(* CoDeSys 2.3 export: TCWIESENRAIN23.EXP *)
(* Libraries: STANDARD.LIB 5.6.98 12:03:02, TcBase.lib 14.5.09 12:14:08, TcEtherCAT.lib 8.3.12 17:06:42, TcSUPS.lib 22.3.10 13:59:22, TcSystem.lib 27.2.12 15:08:36, TcUtilities.lib 10.1.13 20:12:12 *)

(* Task configuration *)
TASK Standard (PRIORITY := 1, INTERVAL := T#10ms);
MAIN
END_TASK
TASK Fast (PRIORITY := 0, INTERVAL := T#1ms);
IO_FAST
END_TASK

(* Global variable list: TwinCAT_Configuration *)
(* Generated automatically by TwinCAT - (read only) *)
VAR_CONFIG
	IO_FAST.uiStateCX5000 AT %IB0 : UINT;
	IO_FAST.uiControlCX5000 AT %QB0 : UINT;
	IO_FAST.iVoltagePhase1 AT %IB2 : ARRAY [0..9] OF INT;	(*  ~ {LinkedWith:TIID^KG-HV A1 X001 (EtherCAT)^KG-HV A35^KG-HV A18^L1 Voltage Samples^U1 SAMPLES} *)
	IO_FAST.iVoltagePhase2 AT %IB22 : ARRAY [0..9] OF INT;	(*  ~ {LinkedWith:TIID^KG-HV A1 X001 (EtherCAT)^KG-HV A35^KG-HV A18^L2 Voltage Samples^U2 SAMPLES} *)
	IO_FAST.iVoltagePhase3 AT %IB42 : ARRAY [0..9] OF INT;	(*  ~ {LinkedWith:TIID^KG-HV A1 X001 (EtherCAT)^KG-HV A35^KG-HV A18^L3 Voltage Samples^U3 SAMPLES} *)
	IO_FAST.uliStartTimeNextLatch AT %IB62 : ARRAY [0..1] OF UDINT;	(*  ~ {LinkedWith:TIID^KG-HV A1 X001 (EtherCAT)^KG-HV A35^KG-HV A18^AI Timestamp NextSync1Time^StartTimeNextLatch} *)
	IO_FAST.bWcState AT %IX72.0 : BOOL;	(*  ~ {LinkedWith:TIID^KG-HV A1 X001 (EtherCAT)^KG-HV A35^KG-HV A18^WcState^WcState} *)
	IO_FAST.fbA28CH1.bRelay AT %QX2.0 : BOOL;	(*  ~ {LinkedWith:TIID^KG-HV A1 K-Bus^KG-HV A1^KG-HV A28^Kanal 1^Ausgang} *)
	IO_FAST.fbA28CH2.bRelay AT %QX2.1 : BOOL;	(*  ~ {LinkedWith:TIID^KG-HV A1 K-Bus^KG-HV A1^KG-HV A28^Kanal 2^Ausgang} *)
	IO_FAST.fbA29CH1.bRelay AT %QX2.2 : BOOL;	(*  ~ {LinkedWith:TIID^KG-HV A1 K-Bus^KG-HV A1^KG-HV A29^Kanal 1^Ausgang} *)
	IO_FAST.fbA29CH2.bRelay AT %QX2.3 : BOOL;	(*  ~ {LinkedWith:TIID^KG-HV A1 K-Bus^KG-HV A1^KG-HV A29^Kanal 2^Ausgang} *)
	IO_FAST.fbA30CH1.bRelay AT %QX2.4 : BOOL;	(*  ~ {LinkedWith:TIID^KG-HV A1 K-Bus^KG-HV A1^KG-HV A30^Kanal 1^Ausgang} *)
	IO_FAST.fbA30CH2.bRelay AT %QX2.5 : BOOL;	(*  ~ {LinkedWith:TIID^KG-HV A1 K-Bus^KG-HV A1^KG-HV A30^Kanal 2^Ausgang} *)
	IO_FAST.fbA31CH1.bRelay AT %QX2.6 : BOOL;	(*  ~ {LinkedWith:TIID^KG-HV A1 K-Bus^KG-HV A1^KG-HV A31^Kanal 1^Ausgang} *)
	IO_FAST.fbA31CH2.bRelay AT %QX2.7 : BOOL;	(*  ~ {LinkedWith:TIID^KG-HV A1 K-Bus^KG-HV A1^KG-HV A31^Kanal 2^Ausgang} *)
	IO_FAST.fbA32CH1.bRelay AT %QX3.0 : BOOL;	(*  ~ {LinkedWith:TIID^KG-HV A1 K-Bus^KG-HV A1^KG-HV A32^Kanal 1^Ausgang} *)
	IO_FAST.fbA32CH2.bRelay AT %QX3.1 : BOOL;	(*  ~ {LinkedWith:TIID^KG-HV A1 K-Bus^KG-HV A1^KG-HV A32^Kanal 2^Ausgang} *)
	IO_FAST.fbA20CH1.bRelay AT %QX3.2 : BOOL;	(*  ~ {LinkedWith:TIID^KG-HV A1 K-Bus^KG-HV A1^KG-HV A20^Kanal 1^KG-Gang Lampe} *)
	IO_FAST.fbA20CH2.bRelay AT %QX3.3 : BOOL;	(*  ~ {LinkedWith:TIID^KG-HV A1 K-Bus^KG-HV A1^KG-HV A20^Kanal 2^KG-EG-Stiege Lampe} *)
	IO_FAST.fbA21CH1.bRelay AT %QX3.4 : BOOL;	(*  ~ {LinkedWith:TIID^KG-HV A1 K-Bus^KG-HV A1^KG-HV A21^Kanal 1^Lager Lampe} *)
	IO_FAST.fbA21CH2.bRelay AT %QX3.5 : BOOL;	(*  ~ {LinkedWith:TIID^KG-HV A1 K-Bus^KG-HV A1^KG-HV A21^Kanal 2^Ausgang} *)
	IO_FAST.fbA23CH1.bRelay AT %QX3.6 : BOOL;	(*  ~ {LinkedWith:TIID^KG-HV A1 K-Bus^KG-HV A1^KG-HV A23^Kanal 1^Heizen Lampe} *)
	IO_FAST.fbA23CH2.bRelay AT %QX3.7 : BOOL;	(*  ~ {LinkedWith:TIID^KG-HV A1 K-Bus^KG-HV A1^KG-HV A23^Kanal 2^WaschenS Lampe} *)
	IO_FAST.fbA24CH1.bRelay AT %QX4.0 : BOOL;	(*  ~ {LinkedWith:TIID^KG-HV A1 K-Bus^KG-HV A1^KG-HV A24^Kanal 1^WaschenN Lampe} *)
	IO_FAST.fbA24CH2.bRelay AT %QX4.1 : BOOL;	(*  ~ {LinkedWith:TIID^KG-HV A1 K-Bus^KG-HV A1^KG-HV A24^Kanal 2^HobbyN Lampe} *)
	IO_FAST.fbA25CH1.bRelay AT %QX4.2 : BOOL;	(*  ~ {LinkedWith:TIID^KG-HV A1 K-Bus^KG-HV A1^KG-HV A25^Kanal 1^Vorrat Lampe} *)
	IO_FAST.fbA25CH2.bRelay AT %QX4.3 : BOOL;	(*  ~ {LinkedWith:TIID^KG-HV A1 K-Bus^KG-HV A1^KG-HV A25^Kanal 2^HobbyS Lampe} *)
	IO_FAST.fbA26CH1.bRelay AT %QX4.4 : BOOL;	(*  ~ {LinkedWith:TIID^KG-HV A1 K-Bus^KG-HV A1^KG-HV A26^Kanal 1^Ausgang} *)
	IO_FAST.fbA26CH2.bRelay AT %QX4.5 : BOOL;	(*  ~ {LinkedWith:TIID^KG-HV A1 K-Bus^KG-HV A1^KG-HV A26^Kanal 2^Ausgang} *)
	IO_FAST.fbA38OGCH1.bRelay AT %QX4.6 : BOOL;
	IO_FAST.fbA38OGCH2.bRelay AT %QX4.7 : BOOL;
	IO_FAST.fbA41OGCH1.bRelay AT %QX5.0 : BOOL;
	IO_FAST.fbA41OGCH2.bRelay AT %QX5.1 : BOOL;
	IO_FAST.fbA43OGCH1.bRelay AT %QX5.2 : BOOL;
	IO_FAST.fbA43OGCH2.bRelay AT %QX5.3 : BOOL;
	IO_FAST.fbA44OGCH1.bRelay AT %QX5.4 : BOOL;
	IO_FAST.fbA44OGCH2.bRelay AT %QX5.5 : BOOL;
	IO_FAST.fbA45OGCH1.bRelay AT %QX5.6 : BOOL;
	IO_FAST.fbA45OGCH2.bRelay AT %QX5.7 : BOOL;
	IO_FAST.fbA48OGCH1.bRelay AT %QX6.0 : BOOL;
	IO_FAST.fbA48OGCH2.bRelay AT %QX6.1 : BOOL;
	IO_FAST.fbA49OGCH1.bRelay AT %QX6.2 : BOOL;
	IO_FAST.fbA49OGCH2.bRelay AT %QX6.3 : BOOL;
	IO_FAST.fbA50OGCH1.bRelay AT %QX6.4 : BOOL;
	IO_FAST.fbA50OGCH2.bRelay AT %QX6.5 : BOOL;
	IO_FAST.fbA52OGCH1.bRelay AT %QX6.6 : BOOL;
	IO_FAST.fbA52OGCH2.bRelay AT %QX6.7 : BOOL;
	IO_FAST.fbA53OGCH1.bRelay AT %QX7.0 : BOOL;
	IO_FAST.fbA53OGCH2.bRelay AT %QX7.1 : BOOL;
	IO_FAST.fbA55OGCH1.bRelay AT %QX7.2 : BOOL;
	IO_FAST.fbA55OGCH2.bRelay AT %QX7.3 : BOOL;
	IO_FAST.fbA56OGCH1.bRelay AT %QX7.4 : BOOL;
	IO_FAST.fbA56OGCH2.bRelay AT %QX7.5 : BOOL;
	IO_FAST.fbA57OGCH1.bRelay AT %QX7.6 : BOOL;
	IO_FAST.fbA57OGCH2.bRelay AT %QX7.7 : BOOL;
	IO_FAST.fbA15OGCH1.bRelay AT %QX8.0 : BOOL;
	IO_FAST.fbA15OGCH2.bRelay AT %QX8.1 : BOOL;
	IO_FAST.fbA17OGCH1.bRelay AT %QX8.2 : BOOL;
	IO_FAST.fbA17OGCH2.bRelay AT %QX8.3 : BOOL;
	IO_FAST.fbA18OGCH1.bRelay AT %QX8.4 : BOOL;
	IO_FAST.fbA18OGCH2.bRelay AT %QX8.5 : BOOL;
	IO_FAST.fbA19OGCH1.bRelay AT %QX8.6 : BOOL;
	IO_FAST.fbA19OGCH2.bRelay AT %QX8.7 : BOOL;
	IO_FAST.fbA21OGCH1.bRelay AT %QX9.0 : BOOL;
	IO_FAST.fbA21OGCH2.bRelay AT %QX9.1 : BOOL;
	IO_FAST.fbA23OGCH1.bRelay AT %QX9.2 : BOOL;
	IO_FAST.fbA23OGCH2.bRelay AT %QX9.3 : BOOL;
	IO_FAST.fbA25OGCH1.bRelay AT %QX9.4 : BOOL;
	IO_FAST.fbA25OGCH2.bRelay AT %QX9.5 : BOOL;
	IO_FAST.fbA26OGCH1.bRelay AT %QX9.6 : BOOL;
	IO_FAST.fbA26OGCH2.bRelay AT %QX9.7 : BOOL;
	IO_FAST.fbA33OGCH1.bRelay AT %QX10.0 : BOOL;
	IO_FAST.fbA33OGCH2.bRelay AT %QX10.1 : BOOL;
	IO_FAST.fbA35OGCH1.bRelay AT %QX10.2 : BOOL;
	IO_FAST.fbA35OGCH2.bRelay AT %QX10.3 : BOOL;
	IO_FAST.fbA36OGCH1.bRelay AT %QX10.4 : BOOL;
	IO_FAST.fbA36OGCH2.bRelay AT %QX10.5 : BOOL;
	IO_FAST.fbA78OGCH1.bRelay AT %QX10.6 : BOOL;
	IO_FAST.fbA78OGCH2.bRelay AT %QX10.7 : BOOL;
	IO_FAST.fbA80OGCH1.bRelay AT %QX11.0 : BOOL;
	IO_FAST.fbA80OGCH2.bRelay AT %QX11.1 : BOOL;
	MAIN._bwmKgGang AT %IX76.0 : BOOL;
	MAIN._tasterHeizen AT %IX76.1 : BOOL;
	MAIN._tasterHobbyL AT %IX76.2 : BOOL;
	MAIN._tasterHobbyR AT %IX76.3 : BOOL;
	MAIN._tasterWaschenL AT %IX76.4 : BOOL;
	MAIN._tasterWaschenR AT %IX76.5 : BOOL;
	MAIN._tasterLagerNO AT %IX76.6 : BOOL;
	MAIN._tasterLagerS AT %IX76.7 : BOOL;
	MAIN._tasterEgGangStiege AT %IX77.0 : BOOL;
	MAIN.heizenHK1.mischer AT %QB12 : INT;
	MAIN.heizenHK1.pumpe AT %QB14 : INT;
	MAIN.heizenHK2.mischer AT %QB16 : INT;
	MAIN.heizenHK2.pumpe AT %QB18 : INT;
END_VAR

(* POU MAIN, ST *)
PROGRAM MAIN
VAR
	ups: FB_S_UPS;
	toggle: FB_Toggle;

	_bwmKgGang AT %I*: BOOL; (* Ost *)
	_tasterHeizen AT %I*: BOOL; (* Sued-West *)
	_tasterHobbyL AT %I*: BOOL; (* Ost *)
	_tasterHobbyR AT %I*: BOOL; (* Ost *)
	_tasterWaschenL AT %I*: BOOL; (* West-Sued *)
	_tasterWaschenR AT %I*: BOOL; (* West-Sued *)
	_tasterLagerNO AT %I*: BOOL;
	_tasterLagerS AT %I*: BOOL;
	_tasterEgGangStiege AT %I*: BOOL; (* Nord *)

	kgGangBwm: FB_Bwm;
	kgGangLicht: FB_Light;

	heizenTaster: FB_Button;
	heizenLicht: FB_Light;
	heizenHK1: FB_Heizkreis;
	heizenHK2: FB_Heizkreis;

	hobbyLichtN: FB_Light;
	hobbyLichtS: FB_Light;

	waschenLichtN: FB_Light;
	waschenLichtS: FB_Light;

	lagerTasterNO: FB_Button;
	lagerTasterS: FB_Button;
	lagerLicht: FB_Light;

	vorratLicht: FB_Light;

	kgEgStiegeLicht: FB_Light;

END_VAR
ups();

(* input processing *)
kgGangBwm(IN := _bwmKgGang, ROOM := 'KG-Gang', LOCATION := 'Ost');
heizenTaster(IN := _tasterHeizen, ROOM := 'Heizen', LOCATION := 'Nord-West');
lagerTasterNO(IN := _tasterLagerNO, ROOM := 'Lager', LOCATION := 'Nord-Ost');
lagerTasterS(IN := _tasterLagerS, ROOM := 'Lager', LOCATION := 'Sued');

(* control *)
toggle(onTime := t#1s, offTime := t#2s);

(* output processing *)
kgGangLicht(IN := kgGangBwm.Q, PT := t#2m);
heizenLicht(IN := heizenTaster.pulseOnClick OR heizentaster.pulseOnLongpress,
	PT := t#15m,
	ROOM := 'Heizen', LOCATION := 'West|Ost');
hobbyLichtS(IN := _tasterHobbyR, PT := t#10m);
waschenLichtN(IN := _tasterWaschenR , PT := t#15m);
waschenLichtS(IN := _tasterWaschenL , PT := t#15m);
lagerLicht(IN := lagerTasterNO.pulseOnClick, FORCE := vorratLicht.Q, FORCE_ON := vorratLicht.Q, PT := t#3m);
vorratLicht(IN := lagerTasterS.pulseOnClick , PT := t#2m);
kgEgStiegeLicht(IN := _tasterEgGangStiege, PT := t#1m);

heizenHk1(soll := 24.0, vorlauf :=, ruecklauf :=);
heizenHk2(soll := 24.0, vorlauf :=, ruecklauf :=);
END_PROGRAM

(* POU FBs/FB_Toggle, ST *)
FUNCTION_BLOCK FB_Toggle
VAR_INPUT
	onTime: TIME :=  t#0.5s;
	offTime: TIME := t#1s;
END_VAR
VAR_OUTPUT
	Q: BOOL;
END_VAR
VAR
	t1: TON;
	t2: TOF;
END_VAR
t1(IN := NOT t2.Q, pt := offTime);
t2(IN := t1.Q, pt := onTime);
Q := t2.Q;
END_FUNCTION_BLOCK

(* POU FBs/FB_Bwm, ST *)
FUNCTION_BLOCK FB_Bwm
VAR_INPUT
	IN: BOOL;
	ROOM: STRING;
	LOCATION: STRING;
END_VAR
VAR_OUTPUT
	Q: BOOL;
END_VAR
Q := IN;
END_FUNCTION_BLOCK

(* POU FBs/FB_Light, ST *)
FUNCTION_BLOCK FB_Light
VAR_INPUT
	IN: BOOL;   (* on/off pulse *)
	PT: TIME;   (* auto-off aka on-time *)
	REACTION: TIME := t#1s;   (* TODO: do not change state right after statechange*)
	FORCE: BOOL;   (* if true, force output on/off, depending on FORCE_ON *)
	FORCE_ON: BOOL;   (* if false and FORCE, then force off *)
	ROOM: STRING;
	LOCATION: STRING;
END_VAR
VAR_OUTPUT RETAIN PERSISTENT
	usageTime: TIME := t#0ms;
	usageDays: UINT := 0;
	usageCounterSwitchOn: UDINT := 0;
END_VAR
VAR_OUTPUT
	Q: BOOL;
END_VAR
VAR
	viText: STRING;
	t: TOF;
	startOpTrigger: R_TRIG;
	stopOpTrigger: F_TRIG;
	opTimetracker: TIME;
	now: TIME;
END_VAR
VAR CONSTANT
	MAX_TIME: TIME := T#71582m47s295ms;
END_VAR
viText := CONCAT(ROOM, '$N');
viText := CONCAT(viText, LOCATION);

IF FORCE THEN
	IF FORCE_ON THEN
		Q := TRUE;
	ELSE
		Q := FALSE;
	END_IF
ELSE (* NOT FORCE *)
	IF IN AND t.Q THEN   (* light on and a signal *)
		(* turn off *)
		t(IN := FALSE, PT := t#0s);
	ELSIF IN AND NOT t.Q THEN   (* light off and a signal *)
		(* turn on *);
		t(IN := IN, PT := PT);
	ELSE (* timer *)
		t(IN := IN, PT := PT);
	END_IF
	Q := t.Q;
END_IF

(* record the operation time *)
startOpTrigger(CLK := Q);
stopOpTrigger(CLK := Q);
IF Q THEN
	now := TIME();
END_IF
IF startOpTrigger.Q THEN
	usageCounterSwitchOn := usageCounterSwitchOn + 1;
	opTimetracker := now;
END_IF
IF Q AND (now < opTimetracker) THEN   (* overflow *)
	usageTime := usageTime + (MAX_TIME - opTimetracker);
	opTimetracker := t#0ms;
END_IF
IF stopOpTrigger.Q THEN
	usageTime := usageTime + (now - opTimetracker);
END_IF
IF Q AND ((now - opTimetracker) > t#1s) THEN
	usageTime := usageTime + (now - opTimetracker);
	opTimetracker := now;
END_IF
IF (Q OR stopOpTrigger.Q) AND (usageTime > t#1d) THEN
	usageDays := usageDays + 1;
	usageTime := usageTime - t#1d;
END_IF
END_FUNCTION_BLOCK

(* POU FBs/FB_Button, ST *)
FUNCTION_BLOCK FB_Button
VAR_INPUT
	ROOM: STRING;
	LOCATION: STRING;
	IN: BOOL;
	LONGPRESS: TIME := t#250ms; (*read by the visualisation*)
END_VAR
VAR_OUTPUT RETAIN PERSISTENT
	isPressed: BOOL := FALSE;
	isLongpressed: BOOL := FALSE;
	isClicked: BOOL := FALSE;
	toggleOnPress: BOOL;
	toggleOnRelease: BOOL;
	toggleOnLongpress: BOOL;
	toggleOnClick: BOOL;
	usageCounterPress: UDINT; (*overall number of press events*)
	usageCounterRelease: UDINT; (*overall number of release events*)
	usageCounterLongpress: UDINT; (*overall number longpress events*)
	usageCounterClick: UDINT; (*overall number of click events*)
END_VAR
VAR_OUTPUT
	isReleased: BOOL; (*NOT isPressed*)
	pulseOnPress: BOOL;
	pulseOnRelease: BOOL;
	pulseOnLongpress: BOOL;
	pulseOnClick: BOOL;
END_VAR
VAR
	viIN: BOOL; (*written by the visualisation*)
	viText: STRING; (*read by the visualisation*)
	pTrig: R_TRIG;
	rTrig: F_TRIG;
	longpressTimer: TON;
	lTrig: R_TRIG;
	cTrig: R_TRIG;
	t1: TOF;
	t2: TOF;
	myIN: BOOL;
END_VAR
(* support VIsualisations *)
viText := CONCAT(ROOM, ' ');
viText := CONCAT(viText, LOCATION);
myIN := IN XOR viIN;

pTrig(CLK := myIN);
rTrig(CLK := myIN);
pulseOnPress := pTrig.Q;
pulseOnRelease := rTrig.Q;

longpressTimer(IN := myIN, PT := LONGPRESS);
lTrig(CLK := longpressTimer.Q);
pulseOnLongpress := ltrig.Q;
IF pulseOnLongpress AND NOT pulseOnRelease THEN
	isLongpressed := TRUE;
	usageCounterLongpress := usageCounterLongpress + 1;
	toggleOnLongpress := fToggle(toggleOnLongpress);
ELSIF pulseOnLongpress THEN
	pulseOnLongpress := FALSE;
END_IF

IF pulseOnPress THEN
	isPressed := TRUE;
	isClicked := FALSE;
	isLongpressed := FALSE;
	usageCounterPress := usageCounterPress + 1;
	toggleOnPress := fToggle(toggleOnPress);
ELSIF pulseOnRelease THEN
	isPressed := FALSE;
	IF isLongpressed THEN
		isLongpressed := FALSE;
	ELSE
		isClicked := TRUE;
		usageCounterClick := usageCounterClick + 1;
		toggleOnClick := fToggle(toggleOnClick);
	END_IF
	usageCounterRelease := usageCounterRelease + 1;
	toggleOnRelease := fToggle(toggleOnRelease);
END_IF
isReleased := NOT isPressed;

cTrig(CLK := isClicked);
pulseOnClick := cTrig.Q;
END_FUNCTION_BLOCK

(* POU Fs/fToggle, ST *)
FUNCTION fToggle : BOOL
VAR_INPUT
	IN: BOOL;
END_VAR
IF IN THEN
	fToggle := FALSE;
ELSE
	fToggle := TRUE;
END_IF
END_FUNCTION

(* POU FBs/FB_Heizkreis, ST *)
FUNCTION_BLOCK FB_Heizkreis
VAR_INPUT
	soll:REAL;
	vorlauf: REAL;
	ruecklauf: REAL;
END_VAR
VAR_OUTPUT
	mischer AT %Q*: INT;   (* 0x7FFF = 100% = 10V; 0x0000 = 0% = 0V*)
	pumpe AT %Q*: INT;   (* 0x7FFF = 100% = 10V; 0x0000 = 0% = 0V*)
END_VAR
VAR
END_VAR
mischer := 6000;
pumpe := 0;
END_FUNCTION_BLOCK

(* POU IO_FAST, ST *)
PROGRAM IO_FAST
VAR
	uiStateCX5000 AT %I*: UINT;
	uiControlCX5000 AT %Q* : UINT;
	iVoltagePhase1 AT %I* : ARRAY [0..9] OF INT;
	iVoltagePhase2 AT %I* : ARRAY [0..9] OF INT;
	iVoltagePhase3 AT %I* : ARRAY [0..9] OF INT;
	uliStartTimeNextLatch AT %I* : ARRAY [0..1] OF UDINT;
	bWcState AT %I* : BOOL;

	fbAnalyseVoltagePhase1 : FB_ANALYSE_VOLTAGE;
	fbAnalyseVoltagePhase2 : FB_ANALYSE_VOLTAGE;
	fbAnalyseVoltagePhase3 : FB_ANALYSE_VOLTAGE;
	fbA28CH1: FB_SYNC_RELAIS;
	fbA28CH2: FB_SYNC_RELAIS;
	fbA29CH1: FB_SYNC_RELAIS;
	fbA29CH2: FB_SYNC_RELAIS;
	fbA30CH1: FB_SYNC_RELAIS;
	fbA30CH2: FB_SYNC_RELAIS;
	fbA31CH1: FB_SYNC_RELAIS;
	fbA31CH2: FB_SYNC_RELAIS;
	fbA32CH1: FB_SYNC_RELAIS;
	fbA32CH2: FB_SYNC_RELAIS;
	fbA20CH1: FB_SYNC_RELAIS;
	fbA20CH2: FB_SYNC_RELAIS;
	fbA21CH1: FB_SYNC_RELAIS;
	fbA21CH2: FB_SYNC_RELAIS;
	fbA23CH1: FB_SYNC_RELAIS;
	fbA23CH2: FB_SYNC_RELAIS;
	fbA24CH1: FB_SYNC_RELAIS;
	fbA24CH2: FB_SYNC_RELAIS;
	fbA25CH1: FB_SYNC_RELAIS;
	fbA25CH2: FB_SYNC_RELAIS;
	fbA26CH1: FB_SYNC_RELAIS;
	fbA26CH2: FB_SYNC_RELAIS;
	fbA38OGCH1: FB_SYNC_RELAIS;
	fbA38OGCH2: FB_SYNC_RELAIS;
	fbA41OGCH1: FB_SYNC_RELAIS;
	fbA41OGCH2: FB_SYNC_RELAIS;
	fbA43OGCH1: FB_SYNC_RELAIS;
	fbA43OGCH2: FB_SYNC_RELAIS;
	fbA44OGCH1: FB_SYNC_RELAIS;
	fbA44OGCH2: FB_SYNC_RELAIS;
	fbA45OGCH1: FB_SYNC_RELAIS;
	fbA45OGCH2: FB_SYNC_RELAIS;
	fbA48OGCH1: FB_SYNC_RELAIS;
	fbA48OGCH2: FB_SYNC_RELAIS;
	fbA49OGCH1: FB_SYNC_RELAIS;
	fbA49OGCH2: FB_SYNC_RELAIS;
	fbA50OGCH1: FB_SYNC_RELAIS;
	fbA50OGCH2: FB_SYNC_RELAIS;
	fbA52OGCH1: FB_SYNC_RELAIS;
	fbA52OGCH2: FB_SYNC_RELAIS;
	fbA53OGCH1: FB_SYNC_RELAIS;
	fbA53OGCH2: FB_SYNC_RELAIS;
	fbA55OGCH1: FB_SYNC_RELAIS;
	fbA55OGCH2: FB_SYNC_RELAIS;
	fbA56OGCH1: FB_SYNC_RELAIS;
	fbA56OGCH2: FB_SYNC_RELAIS;
	fbA57OGCH1: FB_SYNC_RELAIS;
	fbA57OGCH2: FB_SYNC_RELAIS;
	fbA15OGCH1: FB_SYNC_RELAIS;
	fbA15OGCH2: FB_SYNC_RELAIS;
	fbA17OGCH1: FB_SYNC_RELAIS;
	fbA17OGCH2: FB_SYNC_RELAIS;
	fbA18OGCH1: FB_SYNC_RELAIS;
	fbA18OGCH2: FB_SYNC_RELAIS;
	fbA19OGCH1: FB_SYNC_RELAIS;
	fbA19OGCH2: FB_SYNC_RELAIS;
	fbA21OGCH1: FB_SYNC_RELAIS;
	fbA21OGCH2: FB_SYNC_RELAIS;
	fbA23OGCH1: FB_SYNC_RELAIS;
	fbA23OGCH2: FB_SYNC_RELAIS;
	fbA25OGCH1: FB_SYNC_RELAIS;
	fbA25OGCH2: FB_SYNC_RELAIS;
	fbA26OGCH1: FB_SYNC_RELAIS;
	fbA26OGCH2: FB_SYNC_RELAIS;
	fbA33OGCH1: FB_SYNC_RELAIS;
	fbA33OGCH2: FB_SYNC_RELAIS;
	fbA35OGCH1: FB_SYNC_RELAIS;
	fbA35OGCH2: FB_SYNC_RELAIS;
	fbA36OGCH1: FB_SYNC_RELAIS;
	fbA36OGCH2: FB_SYNC_RELAIS;
	fbA78OGCH1: FB_SYNC_RELAIS;
	fbA78OGCH2: FB_SYNC_RELAIS;
	fbA80OGCH1: FB_SYNC_RELAIS;
	fbA80OGCH2: FB_SYNC_RELAIS;


	lrFrequencyPhase1: LREAL;
	lrFrequencyPhase2: LREAL;
	lrFrequencyPhase3: LREAL;
	bErrorL1: BOOL;
	bErrorL2: BOOL;
	bErrorL3: BOOL;
	TON1: TON;
	bStart: BOOL;
	bRelayPLC:BOOL;
END_VAR
(* Spannungsanalyse *)
fbAnalyseVoltagePhase1(
	uliStartTimeNextLatch:=uliStartTimeNextLatch ,
	bWcState:=bWcState ,
	iVoltage:=iVoltagePhase1 ,
	lrFrequency=>lrFrequencyPhase1 ,
	bError=>bErrorL1);

fbAnalyseVoltagePhase2(
	uliStartTimeNextLatch:=uliStartTimeNextLatch ,
	bWcState:=bWcState ,
	iVoltage:=iVoltagePhase2 ,
	lrFrequency=>lrFrequencyPhase2 ,
	bError=>bErrorL2);

fbAnalyseVoltagePhase3(
	uliStartTimeNextLatch:=uliStartTimeNextLatch ,
	bWcState:=bWcState ,
	iVoltage:=iVoltagePhase3 ,
	lrFrequency=>lrFrequencyPhase3 ,
	bError=>bErrorL3);

(* Relais *)
fbA28CH1(bValue:= , udiDelayNanoSek:= 6300000, tNextZeroVoltage:= fbAnalyseVoltagePhase1.tNextZeroVoltage);
fbA28CH2(bValue:= , udiDelayNanoSek:= 7100000, tNextZeroVoltage:= fbAnalyseVoltagePhase1.tNextZeroVoltage);
fbA29CH1(bValue:= , udiDelayNanoSek:= 6800000, tNextZeroVoltage:= fbAnalyseVoltagePhase1.tNextZeroVoltage);
fbA29CH2(bValue:= , udiDelayNanoSek:= 7000000, tNextZeroVoltage:= fbAnalyseVoltagePhase1.tNextZeroVoltage);
fbA30CH1(bValue:= , udiDelayNanoSek:= 7000000, tNextZeroVoltage:= fbAnalyseVoltagePhase1.tNextZeroVoltage);
fbA30CH2(bValue:= , udiDelayNanoSek:= 6200000, tNextZeroVoltage:= fbAnalyseVoltagePhase1.tNextZeroVoltage);
fbA31CH1(bValue:= , udiDelayNanoSek:= 6200000, tNextZeroVoltage:= fbAnalyseVoltagePhase1.tNextZeroVoltage);
fbA31CH2(bValue:= , udiDelayNanoSek:= 6200000, tNextZeroVoltage:= fbAnalyseVoltagePhase1.tNextZeroVoltage);
fbA32CH1(bValue:= , udiDelayNanoSek:= 6500000, tNextZeroVoltage:= fbAnalyseVoltagePhase2.tNextZeroVoltage);
fbA32CH2(bValue:= , udiDelayNanoSek:= 6500000, tNextZeroVoltage:= fbAnalyseVoltagePhase2.tNextZeroVoltage);
fbA20CH1(bValue:= MAIN.kgGangLicht.Q , udiDelayNanoSek:= 7200000, tNextZeroVoltage:= fbAnalyseVoltagePhase1.tNextZeroVoltage);
fbA20CH2(bValue:= MAIN.kgEgStiegeLicht.Q , udiDelayNanoSek:= 6300000, tNextZeroVoltage:= fbAnalyseVoltagePhase1.tNextZeroVoltage);
fbA21CH1(bValue:= MAIN.lagerLicht.Q , udiDelayNanoSek:= 6900000, tNextZeroVoltage:= fbAnalyseVoltagePhase1.tNextZeroVoltage);
fbA21CH2(bValue:= , udiDelayNanoSek:= 7000000, tNextZeroVoltage:= fbAnalyseVoltagePhase1.tNextZeroVoltage);
fbA23CH1(bValue:= MAIN.heizenLicht.Q , udiDelayNanoSek:= 7000000, tNextZeroVoltage:= fbAnalyseVoltagePhase2.tNextZeroVoltage);
fbA23CH2(bValue:= MAIN.waschenLichtS.Q , udiDelayNanoSek:= 6800000, tNextZeroVoltage:= fbAnalyseVoltagePhase2.tNextZeroVoltage);
fbA24CH1(bValue:= MAIN.waschenLichtN.Q , udiDelayNanoSek:= 6800000, tNextZeroVoltage:= fbAnalyseVoltagePhase2.tNextZeroVoltage);
fbA24CH2(bValue:= MAIN.hobbyLichtN.Q, udiDelayNanoSek:= 6500000, tNextZeroVoltage:= fbAnalyseVoltagePhase2.tNextZeroVoltage);
fbA25CH1(bValue:= MAIN.vorratLicht.Q, udiDelayNanoSek:= 6500000, tNextZeroVoltage:= fbAnalyseVoltagePhase2.tNextZeroVoltage);
fbA25CH2(bValue:= MAIN.hobbyLichtS.Q, udiDelayNanoSek:= 6800000, tNextZeroVoltage:= fbAnalyseVoltagePhase2.tNextZeroVoltage);
fbA26CH1(bValue:= , udiDelayNanoSek:= 6800000, tNextZeroVoltage:= fbAnalyseVoltagePhase2.tNextZeroVoltage);
fbA26CH2(bValue:= , udiDelayNanoSek:= 6650000, tNextZeroVoltage:= fbAnalyseVoltagePhase2.tNextZeroVoltage);
fbA38OGCH1(bValue:= , udiDelayNanoSek:= 6500000, tNextZeroVoltage:= fbAnalyseVoltagePhase1.tNextZeroVoltage);
fbA38OGCH2(bValue:= , udiDelayNanoSek:= 6700000, tNextZeroVoltage:= fbAnalyseVoltagePhase1.tNextZeroVoltage);
fbA41OGCH1(bValue:= , udiDelayNanoSek:= 6700000, tNextZeroVoltage:= fbAnalyseVoltagePhase2.tNextZeroVoltage);
fbA41OGCH2(bValue:= , udiDelayNanoSek:= 6100000, tNextZeroVoltage:= fbAnalyseVoltagePhase2.tNextZeroVoltage);
fbA43OGCH1(bValue:= , udiDelayNanoSek:= 6300000, tNextZeroVoltage:= fbAnalyseVoltagePhase1.tNextZeroVoltage);
fbA43OGCH2(bValue:= , udiDelayNanoSek:= 6300000, tNextZeroVoltage:= fbAnalyseVoltagePhase1.tNextZeroVoltage);
fbA44OGCH1(bValue:= , udiDelayNanoSek:= 6300000, tNextZeroVoltage:= fbAnalyseVoltagePhase1.tNextZeroVoltage);
fbA44OGCH2(bValue:= , udiDelayNanoSek:= 6300000, tNextZeroVoltage:= fbAnalyseVoltagePhase1.tNextZeroVoltage);
fbA45OGCH1(bValue:= , udiDelayNanoSek:= 6300000, tNextZeroVoltage:= fbAnalyseVoltagePhase1.tNextZeroVoltage);
fbA45OGCH2(bValue:= , udiDelayNanoSek:= 6300000, tNextZeroVoltage:= fbAnalyseVoltagePhase1.tNextZeroVoltage);
fbA48OGCH1(bValue:= , udiDelayNanoSek:= 6500000, tNextZeroVoltage:= fbAnalyseVoltagePhase2.tNextZeroVoltage);
fbA48OGCH2(bValue:= , udiDelayNanoSek:= 6500000, tNextZeroVoltage:= fbAnalyseVoltagePhase2.tNextZeroVoltage);
fbA49OGCH1(bValue:= , udiDelayNanoSek:= 6500000, tNextZeroVoltage:= fbAnalyseVoltagePhase2.tNextZeroVoltage);
fbA49OGCH2(bValue:= , udiDelayNanoSek:= 6300000, tNextZeroVoltage:= fbAnalyseVoltagePhase2.tNextZeroVoltage);
fbA50OGCH1(bValue:= , udiDelayNanoSek:= 6500000, tNextZeroVoltage:= fbAnalyseVoltagePhase2.tNextZeroVoltage);
fbA50OGCH2(bValue:= , udiDelayNanoSek:= 6100000, tNextZeroVoltage:= fbAnalyseVoltagePhase2.tNextZeroVoltage);
fbA52OGCH1(bValue:= , udiDelayNanoSek:= 6500000, tNextZeroVoltage:= fbAnalyseVoltagePhase2.tNextZeroVoltage);
fbA52OGCH2(bValue:= , udiDelayNanoSek:= 6500000, tNextZeroVoltage:= fbAnalyseVoltagePhase2.tNextZeroVoltage);
fbA53OGCH1(bValue:= , udiDelayNanoSek:= 6400000, tNextZeroVoltage:= fbAnalyseVoltagePhase2.tNextZeroVoltage);
fbA53OGCH2(bValue:= , udiDelayNanoSek:= 6400000, tNextZeroVoltage:= fbAnalyseVoltagePhase2.tNextZeroVoltage);
fbA55OGCH1(bValue:= , udiDelayNanoSek:= 6400000, tNextZeroVoltage:= fbAnalyseVoltagePhase3.tNextZeroVoltage);
fbA55OGCH2(bValue:= , udiDelayNanoSek:= 6100000, tNextZeroVoltage:= fbAnalyseVoltagePhase3.tNextZeroVoltage);
fbA56OGCH1(bValue:= , udiDelayNanoSek:= 6100000, tNextZeroVoltage:= fbAnalyseVoltagePhase3.tNextZeroVoltage);
fbA56OGCH2(bValue:= , udiDelayNanoSek:= 6200000, tNextZeroVoltage:= fbAnalyseVoltagePhase3.tNextZeroVoltage);
fbA57OGCH1(bValue:= , udiDelayNanoSek:= 6100000, tNextZeroVoltage:= fbAnalyseVoltagePhase3.tNextZeroVoltage);
fbA57OGCH2(bValue:= , udiDelayNanoSek:= 6400000, tNextZeroVoltage:= fbAnalyseVoltagePhase3.tNextZeroVoltage);
fbA15OGCH1(bValue:= , udiDelayNanoSek:= 6100000, tNextZeroVoltage:= fbAnalyseVoltagePhase1.tNextZeroVoltage);
fbA15OGCH2(bValue:= , udiDelayNanoSek:= 6300000, tNextZeroVoltage:= fbAnalyseVoltagePhase1.tNextZeroVoltage);
fbA17OGCH1(bValue:= , udiDelayNanoSek:= 6100000, tNextZeroVoltage:= fbAnalyseVoltagePhase2.tNextZeroVoltage);
fbA17OGCH2(bValue:= , udiDelayNanoSek:= 6100000, tNextZeroVoltage:= fbAnalyseVoltagePhase2.tNextZeroVoltage);
fbA18OGCH1(bValue:= , udiDelayNanoSek:= 6100000, tNextZeroVoltage:= fbAnalyseVoltagePhase2.tNextZeroVoltage);
fbA18OGCH2(bValue:= , udiDelayNanoSek:= 6100000, tNextZeroVoltage:= fbAnalyseVoltagePhase2.tNextZeroVoltage);
fbA19OGCH1(bValue:= , udiDelayNanoSek:= 6100000, tNextZeroVoltage:= fbAnalyseVoltagePhase2.tNextZeroVoltage);
fbA19OGCH2(bValue:= , udiDelayNanoSek:= 6100000, tNextZeroVoltage:= fbAnalyseVoltagePhase2.tNextZeroVoltage);
fbA21OGCH1(bValue:= , udiDelayNanoSek:= 6000000, tNextZeroVoltage:= fbAnalyseVoltagePhase3.tNextZeroVoltage);
fbA21OGCH2(bValue:= , udiDelayNanoSek:= 6100000, tNextZeroVoltage:= fbAnalyseVoltagePhase3.tNextZeroVoltage);
fbA23OGCH1(bValue:= , udiDelayNanoSek:= 6100000, tNextZeroVoltage:= fbAnalyseVoltagePhase2.tNextZeroVoltage);
fbA23OGCH2(bValue:= , udiDelayNanoSek:= 6100000, tNextZeroVoltage:= fbAnalyseVoltagePhase2.tNextZeroVoltage);
fbA25OGCH1(bValue:= , udiDelayNanoSek:= 6100000, tNextZeroVoltage:= fbAnalyseVoltagePhase2.tNextZeroVoltage);
fbA25OGCH2(bValue:= , udiDelayNanoSek:= 6100000, tNextZeroVoltage:= fbAnalyseVoltagePhase2.tNextZeroVoltage);
fbA26OGCH1(bValue:= , udiDelayNanoSek:= 6100000, tNextZeroVoltage:= fbAnalyseVoltagePhase2.tNextZeroVoltage);
fbA26OGCH2(bValue:= , udiDelayNanoSek:= 6100000, tNextZeroVoltage:= fbAnalyseVoltagePhase2.tNextZeroVoltage);
fbA33OGCH1(bValue:= , udiDelayNanoSek:= 6100000, tNextZeroVoltage:= fbAnalyseVoltagePhase1.tNextZeroVoltage);
fbA33OGCH2(bValue:= , udiDelayNanoSek:= 6100000, tNextZeroVoltage:= fbAnalyseVoltagePhase1.tNextZeroVoltage);
fbA35OGCH1(bValue:= , udiDelayNanoSek:= 6300000, tNextZeroVoltage:= fbAnalyseVoltagePhase3.tNextZeroVoltage);
fbA35OGCH2(bValue:= , udiDelayNanoSek:= 6200000, tNextZeroVoltage:= fbAnalyseVoltagePhase3.tNextZeroVoltage);
fbA36OGCH1(bValue:= , udiDelayNanoSek:= 6400000, tNextZeroVoltage:= fbAnalyseVoltagePhase3.tNextZeroVoltage);
fbA36OGCH2(bValue:= , udiDelayNanoSek:= 6300000, tNextZeroVoltage:= fbAnalyseVoltagePhase3.tNextZeroVoltage);
fbA78OGCH1(bValue:= , udiDelayNanoSek:= 6300000, tNextZeroVoltage:= fbAnalyseVoltagePhase3.tNextZeroVoltage);
fbA78OGCH2(bValue:= , udiDelayNanoSek:= 6300000, tNextZeroVoltage:= fbAnalyseVoltagePhase3.tNextZeroVoltage);
fbA80OGCH1(bValue:= , udiDelayNanoSek:= 6000000, tNextZeroVoltage:= fbAnalyseVoltagePhase1.tNextZeroVoltage);
fbA80OGCH2(bValue:= , udiDelayNanoSek:= 6000000, tNextZeroVoltage:= fbAnalyseVoltagePhase1.tNextZeroVoltage);
END_PROGRAM

(* POU FBs/FB_ANALYSE_VOLTAGE, ST *)
FUNCTION_BLOCK FB_ANALYSE_VOLTAGE
VAR_INPUT
	uliStartTimeNextLatch : ARRAY [0..1] OF UDINT;
	bWcState		: BOOL;
END_VAR
VAR_IN_OUT
	iVoltage : ARRAY [0..9] OF INT;
END_VAR
VAR
	iBufferV : ARRAY [0..209] OF INT;
	iBufferT : ARRAY [0..209] OF T_DCTIME;
	i: INT;
	dctActSample: T_DCTIME;
	multiplier: T_DCTIME;
	dctSampleDelay: T_DCTIME;
	fbGETCURTASKINDEX: GETCURTASKINDEX;
	tCylceTime: T_DCTIME;
	tSampleTime: T_DCTIME;
	dctElSampleDelta: T_DCTIME;
	n: INT;
	m: INT;
	dctZeroPoint: ARRAY [1..2] OF T_DCTIME;
	bZeroPoint: ARRAY [1..2] OF BOOL;
	ui64Sub: T_ULARGE_INTEGER;
	ui64a: T_ULARGE_INTEGER;
	ui64b: T_ULARGE_INTEGER;
	dctZeroPointDelta: T_DCTIME;
	dctNextSample: T_DCTIME;
	uliStartTimeNextLatchLastCycle: ARRAY [0..1] OF UDINT;
	iBufferZeroSumV: INT;
	dctSampleTimePerV: T_DCTIME;
	dctSampleTimeOffset: T_DCTIME;
	ui64Add: T_ULARGE_INTEGER;
	diResultAdd: DINT;
	diResultSub: DINT;
	ui64Add1: T_ULARGE_INTEGER;
	ui64Sub1: T_ULARGE_INTEGER;
	ui64Cmp1: T_ULARGE_INTEGER;
	iActVoltage: INT;
	tHalfCylceTime: T_DCTIME;
	multi: T_ULARGE_INTEGER;
END_VAR
VAR_OUTPUT
	lrFrequency: LREAL;
	tNextZeroVoltage: T_DCTIME;
	bError: BOOL;
	bZeroFound: BOOL;
	bZeroNow: BOOL;
END_VAR
VAR CONSTANT
	uiOversampling: UINT := 10;
END_VAR
MEMCPY(ADR(dctNextSample), ADR(uliStartTimeNextLatch), SIZEOF(dctActsample));
MEMCPY(ADR(ui64a), ADR(dctNextSample), SIZEOF(ui64a));
MEMCPY(ADR(ui64b), ADR(dctActSample), SIZEOF(ui64b));
ui64Sub := UInt64Sub64(ui64a, ui64b);
MEMCPY(ADR(dctElSampleDelta), ADR(ui64Sub), SIZEOF(dctElSampleDelta));

fbGETCURTASKINDEX(index=> );
tCylceTime.dwLowPart := SYSTEMTASKINFOARR[fbGETCURTASKINDEX.index].cycleTime*100;
tCylceTime.dwHighPart := 0;


IF (dctElSampleDelta.dwLowPart <> tCylceTime.dwLowPart) OR (dctElSampleDelta.dwHighPart <> tCylceTime.dwHighPart) THEN
	bError := TRUE;
ELSE
	bError := FALSE;
END_IF


IF NOT bWcState AND NOT bError THEN
	(* Samplezeit *)
	IF uiOversampling > 0 THEN
		tSampleTime.dwLowPart := (SYSTEMTASKINFOARR[fbGETCURTASKINDEX.index].cycleTime*100)/uiOversampling;
		tSampleTime.dwHighPart := 0;
	END_IF

	(* Spannungsspeicher befüllen *)
	FOR i := 10 TO 209 DO
		iBufferV[i-10] := iBufferV[i];
		iBufferT[i-10] := iBufferT[i];
	END_FOR

	FOR i := 200 TO 209 DO
		multiplier := LREAL_TO_UINT64(INT_TO_LREAL(i-200));
		dctSampleDelay := UInt64Mul64(tSampleTime, multiplier);
		iBufferT[i] := UInt64Add64(dctActSample, dctSampleDelay);
		iBufferV[i] := iVoltage[i-200];
	END_FOR

	(* Zeit der Nulldurchgänge bestimmen *)
	m := 208;
	bZeroPoint[1] := FALSE;
	bZeroPoint[2] := FALSE;
	bZeroNow := FALSE;
	iActVoltage := iBufferV[200];
	FOR n := 1 TO 2 DO
		FOR i := m TO 0 BY -1 DO
			IF (iBufferV[i].15 AND NOT iBufferV[i+1].15) OR (NOT iBufferV[i].15 AND iBufferV[i+1].15) THEN

				iBufferZeroSumV := ABS(iBufferV[i]) + ABS(iBufferV[i+1]);
				IF iBufferZeroSumV > 0 THEN
					dctSampleTimePerV.dwLowPart := LREAL_TO_DWORD(DWORD_TO_LREAL(tSampleTime.dwLowPart) / INT_TO_LREAL(iBufferZeroSumV));
					dctSampleTimePerV.dwHighPart := 0;
					dctSampleTimeOffset := UInt64Mul64(dctSampleTimePerV, LREAL_TO_UINT64(INT_TO_LREAL(ABS(iBufferV[i]))));
					dctZeroPoint[n] := UInt64Add64(iBufferT[i], dctSampleTimeOffset);
				ELSE
					dctZeroPoint[n] := iBufferT[i];
				END_IF


				m := i-1;

				bZeroPoint[n] := TRUE;
				IF n = 1 THEN
					multi.dwLowPart := 1;
					tHalfCylceTime.dwLowPart := tCylceTime.dwLowPart/2;
					ui64Add1 := UInt64Add64(UInt64Add64(dctZeroPoint[n],UInt64Mul64(dctZeroPointDelta, multi)), tHalfCylceTime);
					ui64Sub1 := UInt64Sub64(UInt64Add64(dctZeroPoint[n],UInt64Mul64(dctZeroPointDelta, multi)), tHalfCylceTime);
					ui64Cmp1 := F_GetActualDcTime();
					diResultAdd := UInt64Cmp64(ui64Cmp1, ui64Add1);
					diResultSub := UInt64Cmp64(ui64Cmp1, ui64Sub1);
					IF (diResultSub >= 0) AND (diResultAdd <= 0)THEN
						bZeroNow := TRUE;
					END_IF

				END_IF
				EXIT;
			END_IF
		END_FOR
	END_FOR
	IF bZeroPoint[1] AND bZeroPoint[2] THEN

		(* Berechnung des nächsten Nullpunkts *)
		MEMCPY(ADR(ui64a), ADR(dctZeroPoint[1]), SIZEOF(ui64a));
		MEMCPY(ADR(ui64b), ADR(dctZeroPoint[2]), SIZEOF(ui64b));
		ui64Sub := UInt64Sub64(ui64a, ui64b);
		MEMCPY(ADR(dctZeroPointDelta), ADR(ui64Sub), SIZEOF(dctZeroPointDelta));

		MEMCPY(ADR(ui64a), ADR(dctZeroPointDelta), SIZEOF(ui64a));
		MEMCPY(ADR(ui64b), ADR(dctZeroPoint), SIZEOF(ui64b));
		ui64Add := UInt64Add64(ui64a, ui64b);
		MEMCPY(ADR(tNextZeroVoltage), ADR(ui64Add), SIZEOF(tNextZeroVoltage));


		lrFrequency := 1/(2*DWORD_TO_LREAL(dctZeroPointDelta.dwLowPart)/1000000000);
	END_IF



END_IF
MEMCPY(ADR(dctActSample), ADR(uliStartTimeNextLatch), SIZEOF(dctActsample));

uliStartTimeNextLatchLastCycle := uliStartTimeNextLatch;
END_FUNCTION_BLOCK

(* POU FBs/FB_SYNC_RELAIS, ST *)
FUNCTION_BLOCK FB_SYNC_RELAIS
VAR_INPUT
	bValue : BOOL;
	udiDelayNanoSek : UDINT;
	tNextZeroVoltage: T_DCTIME;
END_VAR
VAR_OUTPUT
	bRelay AT %Q* : BOOL;
END_VAR
VAR
	fbGETCURTASKINDEX: GETCURTASKINDEX;
	tNextZeroVoltageLast: T_DCTIME;
	TON_FAILURE: TON;
	TOF_WAIT: TOF;
	udiLastOnlineChangeCount: UDINT;
	multi: T_DCTIME;
	ui64Add1: T_ULARGE_INTEGER;
	tHalfCylceTime: T_DCTIME;
	ui64Sub1: T_ULARGE_INTEGER;
	ui64Cmp1: T_ULARGE_INTEGER;
	diResultAdd: DINT;
	diResultSub: DINT;
	tCylceTime: T_DCTIME;
END_VAR
(*fTvalue(CLK:=bValue AND bRelay);
IF fTvalue.Q OR bReset THEN
	bRelay := FALSE;
	bReset := FALSE;
END_IF
*)
TON_FAILURE(IN:=tNextZeroVoltage.dwLowPart = tNextZeroVoltageLast.dwLowPart, PT:=t#100ms);
tNextZeroVoltageLast.dwLowPart := tNextZeroVoltage.dwLowPart;

TOF_WAIT(IN:=SYSTEMINFO.onlineChangeCount <> udiLastOnlineChangeCount, PT:= t#0.5s);
udiLastOnlineChangeCount := SYSTEMINFO.onlineChangeCount;



IF bValue AND NOT bRelay AND NOT TON_FAILURE.Q THEN
	fbGETCURTASKINDEX(index=> );
	tCylceTime.dwLowPart := SYSTEMTASKINFOARR[fbGETCURTASKINDEX.index].cycleTime*100;
	tCylceTime.dwHighPart := 0;

	multi.dwLowPart := udiDelayNanoSek;
	tHalfCylceTime.dwLowPart := tCylceTime.dwLowPart/2;
	ui64Add1 := UInt64Add64(UInt64Sub64(tNextZeroVoltage,multi), tHalfCylceTime);
	ui64Sub1 := UInt64Sub64(UInt64Sub64(tNextZeroVoltage,multi), tHalfCylceTime);
	ui64Cmp1 := F_GetActualDcTime();
	diResultAdd := UInt64Cmp64(ui64Cmp1, ui64Add1);
	diResultSub := UInt64Cmp64(ui64Cmp1, ui64Sub1);

	IF (diResultSub >= 0) AND (diResultAdd <= 0)THEN
		bRelay := TRUE;
	END_IF
END_IF

IF NOT bValue AND bRelay AND NOT TON_FAILURE.Q THEN
	fbGETCURTASKINDEX(index=> );
	tCylceTime.dwLowPart := SYSTEMTASKINFOARR[fbGETCURTASKINDEX.index].cycleTime*100;
	tCylceTime.dwHighPart := 0;

	multi.dwLowPart := udiDelayNanoSek/2;
	tHalfCylceTime.dwLowPart := tCylceTime.dwLowPart/2;
	ui64Add1 := UInt64Add64(UInt64Sub64(tNextZeroVoltage,multi), tHalfCylceTime);
	ui64Sub1 := UInt64Sub64(UInt64Sub64(tNextZeroVoltage,multi), tHalfCylceTime);
	ui64Cmp1 := F_GetActualDcTime();
	diResultAdd := UInt64Cmp64(ui64Cmp1, ui64Add1);
	diResultSub := UInt64Cmp64(ui64Cmp1, ui64Sub1);

	IF (diResultSub >= 0) AND (diResultAdd <= 0)THEN
		bRelay := FALSE;
	END_IF
END_IF
END_FUNCTION_BLOCK

(* Visualisation HEIZEN
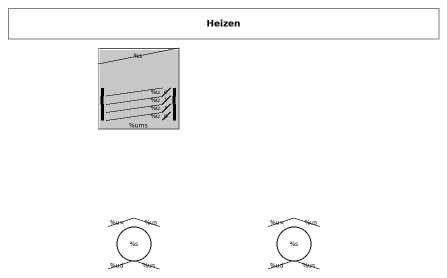
embedded screen at (280,50)-(361,131): viButtonSingle
embedded screen at (290,220)-(341,271): viLight; dynamic style MAIN.viHeizenLicht
embedded screen at (450,220)-(501,271): viLight
rounded rectangle at (190,10)-(621,41): text "Heizen"
*)

(* Visualisation Hobby
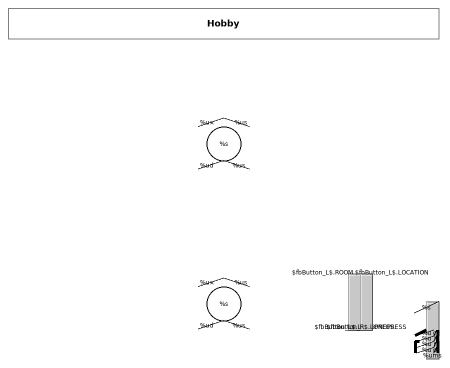
embedded screen at (380,120)-(431,171): viLight
rounded rectangle at (190,10)-(621,41): text "Hobby"
embedded screen at (380,280)-(431,331): viLight
embedded screen at (530,270)-(621,361): viButtonDouble
*)

(* Visualisation KG
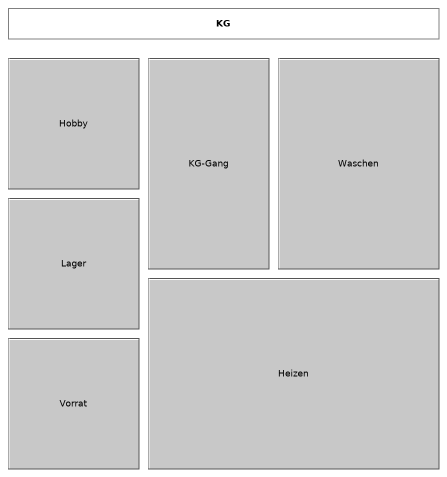
button at (330,280)-(621,471): text "Heizen"; opens Heizen
button at (190,340)-(321,471): text "Vorrat"; opens Vorrat
button at (190,200)-(321,331): text "Lager"; opens Lager
button at (190,60)-(321,191): text "Hobby"; opens Hobby
button at (460,60)-(621,271): text "Waschen"; opens Waschen
rounded rectangle at (190,10)-(621,41): text "KG"
button at (330,60)-(451,271): text "KG-Gang"; opens KG-Gang
*)

(* Visualisation LAGER
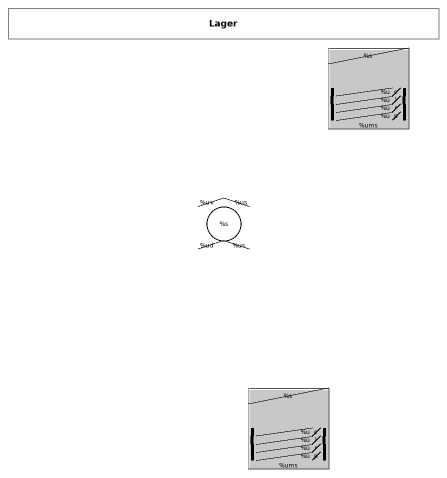
embedded screen at (510,50)-(591,131): viButtonSingle
embedded screen at (380,200)-(431,251): viLight
rounded rectangle at (190,10)-(621,41): text "Lager"
embedded screen at (430,390)-(511,471): viButtonSingle
*)

(* Visualisation VORRAT
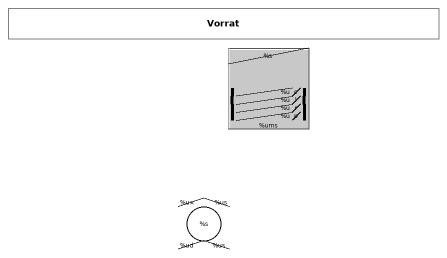
embedded screen at (360,200)-(411,251): viLight
rounded rectangle at (190,10)-(621,41): text "Vorrat"
embedded screen at (410,50)-(491,131): viButtonSingle
*)

(* Visualisation Waschen
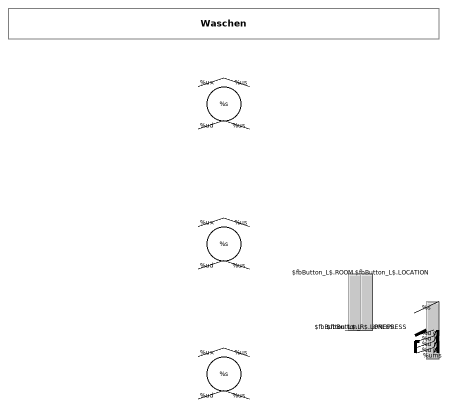
embedded screen at (380,80)-(431,131): viLight
rounded rectangle at (190,10)-(621,41): text "Waschen"
embedded screen at (380,220)-(431,271): viLight
embedded screen at (530,270)-(621,361): viButtonDouble
embedded screen at (380,350)-(431,401): viLight
*)

(* Visualisation viButtonDouble
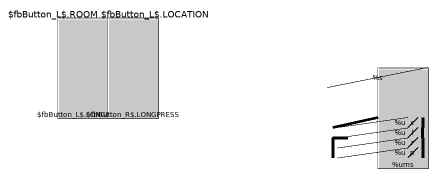
button at (0,10)-(51,111): text "$fbButton_L$.LONGPRESS"; taps $fbButton_L$.IN
button at (50,10)-(101,111): text "$fbButton_R$.LONGPRESS"; taps $fbButton_R$.IN
rectangle at (0,0)-(101,11): text "$fbButton_L$.ROOM $fbButton_L$.LOCATION"
button at (320,60)-(371,161): text "%ums"; shows $fbButton$.LONGPRESS; taps $fbButton$.viIN
curve at (270,60)-(370,80): text "%s"; shows $fbButton$.viText
curve at (280,140)-(350,150): text "%u"; shows $fbButton$.usageCounterPress
curve at (365,140)-(365,150): alarm colour if $fbButton$.toggleOnPress
curve at (365,130)-(365,140): alarm colour if $fbButton$.toggleOnRelease
curve at (365,120)-(365,130): alarm colour if $fbButton$.toggleOnLongpress
curve at (365,110)-(365,120): alarm colour if $fbButton$.toggleOnClick
curve at (280,130)-(350,140): text "%u"; shows $fbButton$.usageCounterRelease
curve at (280,120)-(350,130): text "%u"; shows $fbButton$.usageCounterLongpress
curve at (280,110)-(350,120): text "%u"; shows $fbButton$.usageCounterClick
curve at (350,110)-(360,120): text "c"
curve at (350,120)-(360,130): text "l"
curve at (350,130)-(360,140): text "r"
curve at (350,140)-(360,150): text "p"
curve at (275,140)-(275,150): alarm colour if $fbButton$.isPressed
curve at (275,130)-(275,140): alarm colour if $fbButton$.isReleased
curve at (275,130)-(290,130): alarm colour if $fbButton$.isLongpressed
curve at (275,110)-(320,120): alarm colour if $fbButton$.isClicked
*)

(* Visualisation viButtonSingle
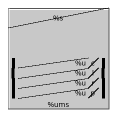
button at (0,0)-(101,101): text "%ums"; shows $fbButton$.LONGPRESS; taps $fbButton$.viIN
curve at (0,0)-(100,20): text "%s"; shows $fbButton$.viText
curve at (10,80)-(80,90): text "%u"; shows $fbButton$.usageCounterPress
curve at (95,80)-(95,90): alarm colour if $fbButton$.toggleOnPress
curve at (95,70)-(95,80): alarm colour if $fbButton$.toggleOnRelease
curve at (95,60)-(95,70): alarm colour if $fbButton$.toggleOnLongpress
curve at (95,50)-(95,60): alarm colour if $fbButton$.toggleOnClick
curve at (10,70)-(80,80): text "%u"; shows $fbButton$.usageCounterRelease
curve at (10,60)-(80,70): text "%u"; shows $fbButton$.usageCounterLongpress
curve at (10,50)-(80,60): text "%u"; shows $fbButton$.usageCounterClick
curve at (80,50)-(90,60): text "c"
curve at (80,60)-(90,70): text "l"
curve at (80,70)-(90,80): text "r"
curve at (80,80)-(90,90): text "p"
curve at (5,80)-(5,90): alarm colour if $fbButton$.isPressed
curve at (5,70)-(5,80): alarm colour if $fbButton$.isReleased
curve at (5,60)-(5,70): alarm colour if $fbButton$.isLongpressed
curve at (5,50)-(5,60): alarm colour if $fbButton$.isClicked
*)

(* Visualisation viButtonTripple
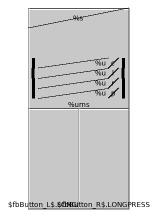
button at (0,0)-(101,101): text "%ums"; shows $fbButton_T$.LONGPRESS; taps $fbButton_T$.viIN
button at (0,100)-(51,201): text "$fbButton_L$.LONGPRESS"; taps $fbButton_L$.IN
button at (50,100)-(101,201): text "$fbButton_R$.LONGPRESS"; taps $fbButton_R$.IN
curve at (0,0)-(100,20): text "%s"; shows $fbButton_T$.viText
curve at (10,80)-(80,90): text "%u"; shows $fbButton_T$.usageCounterPress
curve at (95,80)-(95,90): alarm colour if $fbButton_T$.toggleOnPress
curve at (95,70)-(95,80): alarm colour if $fbButton_T$.toggleOnRelease
curve at (95,60)-(95,70): alarm colour if $fbButton_T$.toggleOnLongpress
curve at (95,50)-(95,60): alarm colour if $fbButton_T$.toggleOnClick
curve at (10,70)-(80,80): text "%u"; shows $fbButton_T$.usageCounterRelease
curve at (10,60)-(80,70): text "%u"; shows $fbButton_T$.usageCounterLongpress
curve at (10,50)-(80,60): text "%u"; shows $fbButton_T$.usageCounterClick
curve at (80,50)-(90,60): text "c"
curve at (80,60)-(90,70): text "l"
curve at (80,70)-(90,80): text "r"
curve at (80,80)-(90,90): text "p"
curve at (5,80)-(5,90): alarm colour if $fbButton_T$.isPressed
curve at (5,70)-(5,80): alarm colour if $fbButton_T$.isReleased
curve at (5,60)-(5,70): alarm colour if $fbButton_T$.isLongpressed
curve at (5,50)-(5,60): alarm colour if $fbButton_T$.isClicked
*)

(* Visualisation viLight
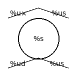
ellipse at (10,10)-(51,51): invisible if NOT $fbLight$.FORCE
ellipse at (10,10)-(51,51): text "%s"; shows $fbLight$.viText; alarm colour if $fbLight$.Q
curve at (30,50)-(60,60): text "%us"; shows $fbLight$.usageTime / 1000
curve at (0,50)-(30,60): text "%ud"; shows $fbLight$.usageDays
curve at (0,0)-(30,10): text "%u×"; shows $fbLight$.usageCounterSwitchOn
curve at (30,0)-(60,10): text "%us"; shows ($fbLight$.PT - $fbLight$.t.ET) / 1000
*)

(* Visualisation MAIN
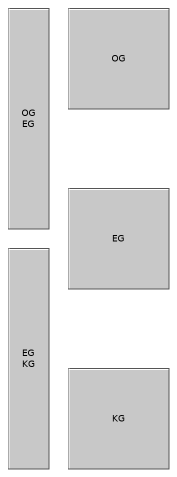
button at (70,370)-(171,471): text "KG"; opens KG
button at (70,190)-(171,291): text "EG"; opens EG
button at (70,10)-(171,111): text "OG"; opens OG
button at (10,250)-(51,471): text "EG / KG"; opens KG-EG
button at (10,10)-(51,231): text "OG / EG"; opens EG-OG
*)
